Omron CX-Programmer project NewProject (CX-Programmer 9.61)

# PLC NewPLC1: CPM2* 

## Program NewProgram1 (no task)

### Section Section1

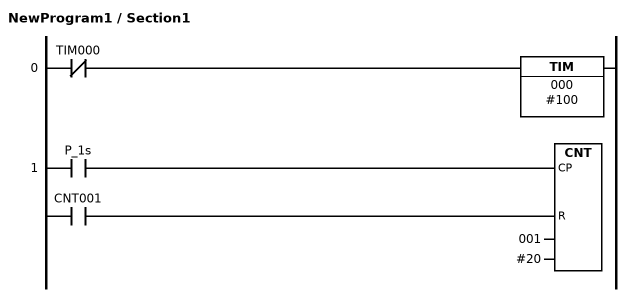
; rung 0
LDNOT TIM000
TIM 000 #100
; rung 1
LD P_1s
LD CNT001
CNT 001 #20

### Section Section2
; rung 0
END(01)